TYPE ST_MinMax :
STRUCT
	lrMin: LREAL;
	lrMax: LREAL;
END_STRUCT
END_TYPE

(* stored: Version 1.1.0.1, ProductVersion 3.1.4020.6
   DUT ST_MinMax: Id {7822ab5a-e746-468d-bd91-2eaa28e24418} *)
